FUNCTION_BLOCK fbPiston EXTENDS TcoCore.TcoComponent
VAR_INPUT
	iHomePositionSensor : BOOL;
	iWorkPositionSensor : BOOL;	
END_VAR

VAR_OUTPUT
	qHomePositionActuator : BOOL;
	qWorkPositionActuator : BOOL;		
END_VAR

VAR
	_moveHomeTask : fbPistonMoveTask(THIS^);
	_moveWorkTask : fbPistonMoveTask(THIS^);
END_VAR

_moveHomeTask(PositionSensor := iHomePositionSensor, MoveToPositionSignal := qHomePositionActuator, InverseSignal := qWorkPositionActuator);
_moveWorkTask(PositionSensor := iWorkPositionSensor, MoveToPositionSignal := qWorkPositionActuator, InverseSignal := qHomePositionActuator);

METHOD PROTECTED Manual
VAR_INPUT
END_VAR
END_METHOD

METHOD MoveHome : TcoCore.ITcoTask
MoveHome := THIS^._moveHomeTask.Invoke();
END_METHOD

METHOD MoveWork : TcoCore.ITcoTask
MoveWork := THIS^._moveWorkTask.Invoke();
END_METHOD

METHOD  Restore : ITcoRestorable
THIS^._moveHomeTask.Restore();
THIS^._moveWorkTask.Restore();
END_METHOD

END_FUNCTION_BLOCK

(* stored: Version 1.1.0.1, ProductVersion 3.1.4024.6
   POU fbPiston: Id {c4094ed5-4fe0-0f6e-24e6-4cc0fa53181e}, SpecialFunc None
   Method Manual: Id {e2305248-08d3-0a45-0227-6f8abe0d86d9}
   Method MoveHome: Id {ec08a57d-3edb-01f0-35bc-3c8a96242bb9}
   Method MoveWork: Id {e9e0be0c-566d-0749-1c75-1097c8dadecf}
   Method Restore: Id {fc7ee28d-fd88-0b69-144e-14e0b2374ab2} *)
